FUNCTION F_LrSecond2Time : Time
VAR_INPUT
	lrSecond	: LREAL;
END_VAR
VAR
END_VAR

F_LrSecond2Time := lreal_to_time(lrSecond*1000);

END_FUNCTION

(* stored: Version 1.1.0.1, ProductVersion 3.1.4024.12
   POU F_LrSecond2Time: Id {163fab69-9968-486a-b1cd-5f54df0942a0}, SpecialFunc None *)
